// Implicitly generated code : DO NOT EDIT
FUNCTION CheckDivReal : REAL
VAR_INPUT
	divisor:REAL;
END_VAR

// Implicitly generated code : Only an Implementation suggestion
{noflow}
Fault_Count_G(CU:=FALSE) ; 
IF divisor = 0 THEN
	CheckDivReal:=1;
		Fault_Count_G(CU:=TRUE) ; 
ELSE
	CheckDivReal:=divisor;
END_IF;
{flow}

END_FUNCTION

(* stored: Version 1.1.0.1, ProductVersion 3.1.4024.2
   POU CheckDivReal: Id {585a9b27-0b6d-4072-8940-64595e27f587}, SpecialFunc CheckDivReal32 *)
